FUNCTION F_Throughput : UDINT
VAR_INPUT
    nCaps        : UDINT;
    nCycleTimeMs : UDINT;
END_VAR

F_Throughput := nCaps * 60000 / nCycleTimeMs;

END_FUNCTION

(* stored: Version 1.1.0.1, ProductVersion 3.1.4024.0
   POU F_Throughput: Id {b04ec53f-be06-4952-b240-d2b3b69ffc8f}, SpecialFunc None *)
